ABB RAPID module: Module1.mod

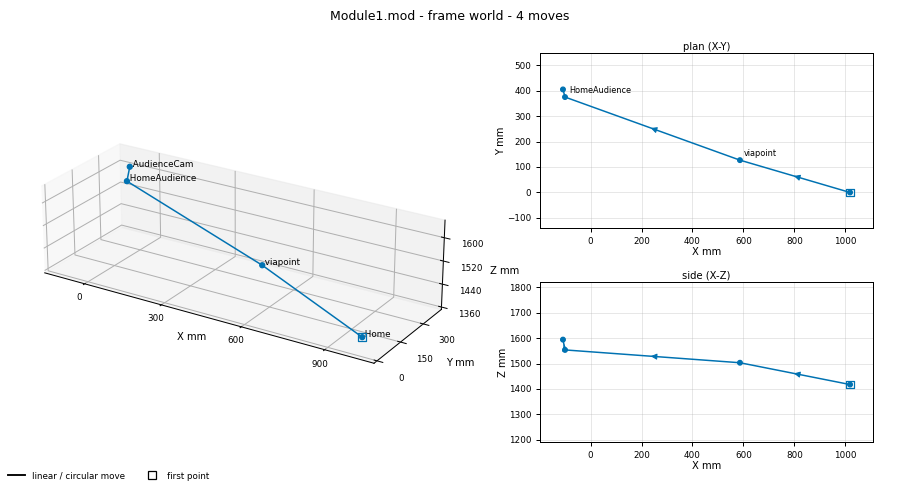
[picture p0: tool path of Module1.mod in frame world, 4 of 4 moves have a stored position in this frame; points joined in program order, loops and branches not executed]
MODULE Module1
    CONST robtarget AboveDuster:=[[743.879676977,-800.509897995,1300.071035327],[0.000000006,0.382683505,0.923879502,0.000000013],[-1,0,-2,0],[9E+09,9E+09,9E+09,9E+09,9E+09,9E+09]];
    CONST robtarget Duster:=[[743.879739272,-800.509937926,866.646225387],[0,0.382683433,0.923879532,0],[-1,0,-2,0],[9E+09,9E+09,9E+09,9E+09,9E+09,9E+09]];
    CONST robtarget Home:=[[1018.612159322,0,1417.5],[0.5,0,0.866025404,0],[0,0,0,0],[9E+09,9E+09,9E+09,9E+09,9E+09,9E+09]];
    CONST robtarget AudienceCam:=[[-108.392054445,404.524654327,1593.865850606],[0.306068712,-0.601521785,0.556041018,0.48508955],[1,-1,0,0],[9E+09,9E+09,9E+09,9E+09,9E+09,9E+09]];
    CONST robtarget HomeAudience:=[[-100.362523078,374.558223054,1553.37723237],[0.160813199,-0.7001828,0.647242369,0.254873454],[1,0,0,0],[9E+09,9E+09,9E+09,9E+09,9E+09,9E+09]];
    CONST robtarget viapoint:=[[586.472283508,126.846671607,1503.046845036],[0.572111865,-0.33163658,0.740341252,-0.120830555],[0,-1,-1,0],[9E+09,9E+09,9E+09,9E+09,9E+09,9E+09]];
    CONST robtarget AbovePen:=[[986.400074312,794.700007103,1226.400174056],[-0.000000007,-0.35720179,0.934027238,-0.000000002],[0,0,-1,0],[9E+09,9E+09,9E+09,9E+09,9E+09,9E+09]];
    PROC AudienceCamPath()
        MoveL Home,v1000,fine,tool0\WObj:=wobj0;
        MoveL viapoint,v1000,z100,tool0\WObj:=wobj0;
        MoveL HomeAudience,v1000,z100,tool0\WObj:=wobj0;
        MoveL AudienceCam,v1000,fine,tool0\WObj:=wobj0;
    ENDPROC
ENDMODULE
